FUNCTION_BLOCK SERVO_POS_CONFIRM
VAR_INPUT
	BOOL_JOG_ACTIVE : BOOL;
	UINT_TARGET1 : UINT;
	UINT_TARGET2 : UINT;
	UINT_TARGET3 : UINT;
	UINT_TARGET4 : UINT;
	COUNTER_VALUE : UINT;
	HOMING_READY : BOOL;
END_VAR

VAR_OUTPUT
	TARGET1_CONFIRM_BOOL : BOOL;
	TARGET2_CONFIRM_BOOL : BOOL;
	TARGET3_CONFIRM_BOOL : BOOL;
	TARGET4_CONFIRM_BOOL : BOOL;
END_VAR
VAR
	T1C: BOOL;
	T2C: BOOL;
	T3C: BOOL;
	T4C: BOOL;
END_VAR

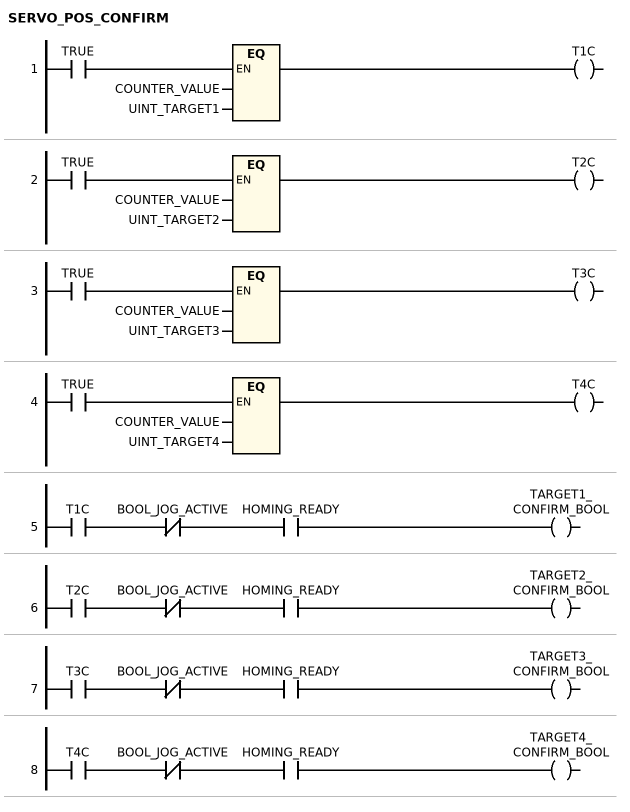
// NETWORK 1
T1C := COUNTER_VALUE = UINT_TARGET1;

// NETWORK 2
T2C := COUNTER_VALUE = UINT_TARGET2;

// NETWORK 3
T3C := COUNTER_VALUE = UINT_TARGET3;

// NETWORK 4
T4C := COUNTER_VALUE = UINT_TARGET4;

// NETWORK 5
TARGET1_CONFIRM_BOOL := T1C AND NOT BOOL_JOG_ACTIVE AND HOMING_READY;

// NETWORK 6
TARGET2_CONFIRM_BOOL := T2C AND NOT BOOL_JOG_ACTIVE AND HOMING_READY;

// NETWORK 7
TARGET3_CONFIRM_BOOL := T3C AND NOT BOOL_JOG_ACTIVE AND HOMING_READY;

// NETWORK 8
TARGET4_CONFIRM_BOOL := T4C AND NOT BOOL_JOG_ACTIVE AND HOMING_READY;

END_FUNCTION_BLOCK

(* stored: Version 1.1.0.1, ProductVersion 3.1.4024.12
   POU SERVO_POS_CONFIRM: Id {996c49a1-50fa-4023-b316-d502fad7d297}, SpecialFunc None *)
